PROGRAM Ax_01_AxisMoveAbsRel_06
VAR
	HMI_Motion: FB_HMI_Control_NoGroupRef;


	tMessageOffset: UINT;
	tNumMessagesPerRow: UINT;
	
	
	MyAdvanceInterlock: BOOL;
	MyReturnInterlock: BOOL;
	
	MyAutoAdvanceCondition: BOOL;
	MyAutoReturnCondition: BOOL;
	
	myAdvancePrompt: BOOL;
	myReturnPrompt: BOOL;
	

	NotUsed: UINT;

END_VAR

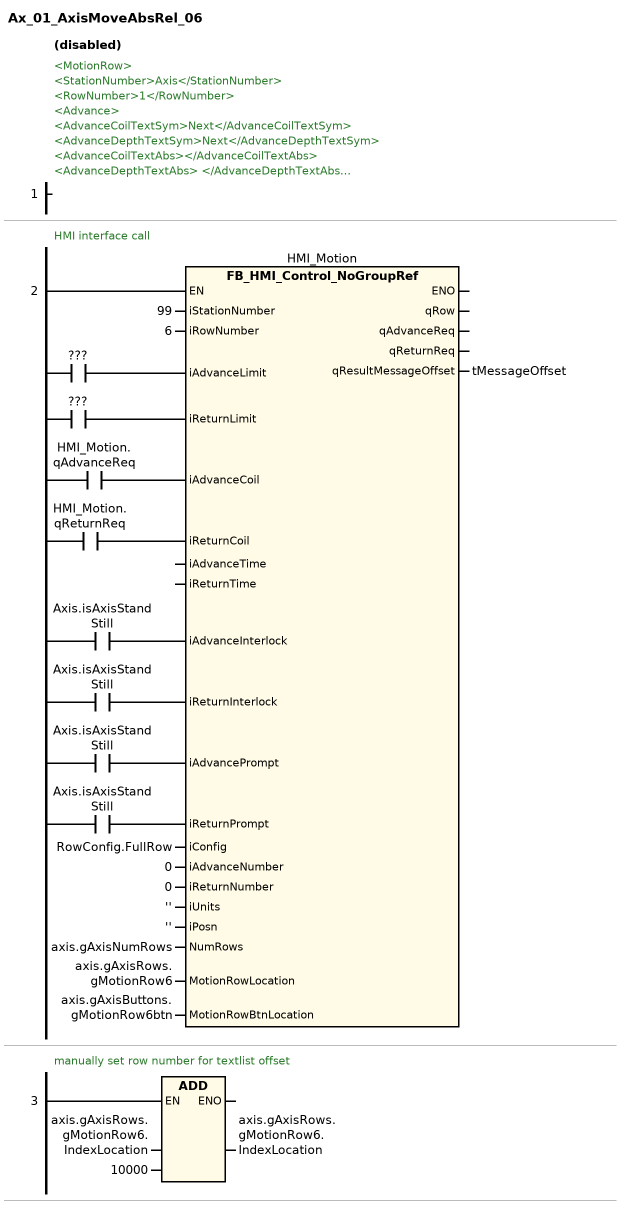
// NETWORK 1 (disabled)
// <MotionRow>
// <StationNumber>Axis</StationNumber>
// <RowNumber>1</RowNumber>
//   <Advance>
//     <AdvanceCoilTextSym>Next</AdvanceCoilTextSym>
//     <AdvanceDepthTextSym>Next</AdvanceDepthTextSym>
//     <AdvanceCoilTextAbs></AdvanceCoilTextAbs>
//     <AdvanceDepthTextAbs> </AdvanceDepthTextAbs>
//     <ManSeq></ManSeq>
//   </Advance>
//   <Return>
//     <ReturnCoilTextSym>Previous</ReturnCoilTextSym>
//     <ReturnDepthTextSym>Previous</ReturnDepthTextSym>
//     <ReturnCoilTextAbs></ReturnCoilTextAbs>
//     <ReturnDepthTextAbs></ReturnDepthTextAbs>
//    <ManSeq></ManSeq>
//   </Return>
//   <Motion>
//     <NameSym>Axis Name</NameSym>
//     <NameAbs>X1</NameAbs>
//   </Motion>
// </MotionRow>

// NETWORK 2
// HMI interface call
HMI_Motion(
    iStationNumber := 99,
    iRowNumber := 6,
    iAdvanceCoil := HMI_Motion.qAdvanceReq,
    iReturnCoil := HMI_Motion.qReturnReq,
    iAdvanceInterlock := Axis.isAxisStandStill,
    iReturnInterlock := Axis.isAxisStandStill,
    iAdvancePrompt := Axis.isAxisStandStill,
    iReturnPrompt := Axis.isAxisStandStill,
    iConfig := RowConfig.FullRow,
    iAdvanceNumber := 0,
    iReturnNumber := 0,
    iUnits := '',
    iPosn := '',
    NumRows := axis.gAxisNumRows,
    MotionRowLocation := axis.gAxisRows.gMotionRow6,
    MotionRowBtnLocation := axis.gAxisButtons.gMotionRow6btn,
    qResultMessageOffset => tMessageOffset); // FB_HMI_Control_NoGroupRef

// NETWORK 3
// manually set row number for textlist offset
axis.gAxisRows.gMotionRow6.IndexLocation := axis.gAxisRows.gMotionRow6.IndexLocation + 10000;

END_PROGRAM

(* stored: Version 1.1.0.1, ProductVersion 3.1.4024.12
   POU Ax_01_AxisMoveAbsRel_06: Id {f8a203fd-7b17-4e4a-ac83-f29116baa21b}, SpecialFunc None *)
